{attribute 'c++_compatible'}
// class for implementing IotWebSocetClient functions without exposing them may only be used for ARCommunication_t
FUNCTION_BLOCK ARCommunicationWSExtentionWS_t EXTENDS FB_IotWebSocketClient
VAR_INPUT
END_VAR
VAR_OUTPUT
	lastMessage : STRING(255) := ''; // last recived message
END_VAR
VAR	
	_newMessageAvalable : BOOL := FALSE; // is set true whenever a new message arrives
END_VAR

PROPERTY newMessageAvalable : bool
GET
newMessageAvalable :=  _newMessageAvalable;
END_GET
SET
_newMessageAvalable := newMessageAvalable;
END_SET
END_PROPERTY

{attribute 'TcTypeSystem'}
{attribute 'c++_compatible'}
{attribute 'minimal_input_size' := '4'}
{attribute 'pack_mode' := '4'}
{attribute 'TcRpcEnable'}
METHOD OnWebSocketClose : Global.HRESULT
VAR_INPUT
	statusCode	: UINT;
	content	: Global.PVOID;
	contentLength	: UDINT;
END_VAR
END_METHOD

{attribute 'TcTypeSystem'}
{attribute 'c++_compatible'}
{attribute 'minimal_input_size' := '4'}
{attribute 'pack_mode' := '4'}
{attribute 'TcRpcEnable'}
METHOD OnWebSocketMessage : Global.HRESULT
VAR_INPUT
	content	: Global.PVOID;
	contentLength	: UDINT;
	contentType	: Global.ETcIotWebSocketContentType;
END_VAR
VAR
	ptr : POINTER TO STRING;
END_VAR
// if it isn't text, drop packet
IF  contentType = Global.ETcIotWebSocketContentType.WS_CONTENT_TEXT THEN
		ptr := content;
		THIS^.lastMessage := ptr^;
		THIS^._newMessageAvalable := TRUE;	
END_IF
END_METHOD

{attribute 'TcTypeSystem'}
{attribute 'c++_compatible'}
{attribute 'minimal_input_size' := '4'}
{attribute 'pack_mode' := '4'}
{attribute 'TcRpcEnable'}
METHOD OnWebSocketOpen : Global.HRESULT
VAR_IN_OUT CONSTANT
	webSocketProtocol	: STRING;
	origin	: STRING;
END_VAR
VAR_INPUT
	bPerMessageDeflate	: BOOL;
END_VAR
END_METHOD

{attribute 'TcTypeSystem'}
{attribute 'c++_compatible'}
{attribute 'minimal_input_size' := '4'}
{attribute 'pack_mode' := '4'}
METHOD TcAddRef : UDINT
END_METHOD

{attribute 'TcTypeSystem'}
{attribute 'c++_compatible'}
{attribute 'minimal_input_size' := '4'}
{attribute 'pack_mode' := '4'}
METHOD TcQueryInterface : Global.HRESULT
VAR_INPUT
	iid	: REFERENCE TO Global.IID;
	pipItf	: POINTER TO Global.PVOID;
END_VAR
END_METHOD

{attribute 'TcTypeSystem'}
{attribute 'c++_compatible'}
{attribute 'minimal_input_size' := '4'}
{attribute 'pack_mode' := '4'}
METHOD TcRelease : UDINT
END_METHOD

END_FUNCTION_BLOCK

(* stored: Version 1.1.0.1
   POU ARCommunicationWSExtentionWS_t: Id {b160b582-710e-48ca-a2e1-674bfaf42c51}, SpecialFunc None
   Property newMessageAvalable: Id {60cc030d-e252-40bf-962d-546e21880d27}
   Get Get: Id {89613a16-3d29-4b2d-8a2e-e805c75c660f}
   Set Set: Id {d84cd38f-e2d7-45a5-a66d-f3b744e69d9f}
   Method OnWebSocketClose: Id {83b963f1-cb68-4c4f-839b-6fe0c3279a4b}
   Method OnWebSocketMessage: Id {aafc85e2-e4b6-4b40-a50f-be62207a97c2}
   Method OnWebSocketOpen: Id {84b70aa8-e731-4dfb-b3ce-e492968de315}
   Method TcAddRef: Id {19906943-71ba-4126-b01d-557cf40c9802}
   Method TcQueryInterface: Id {591f8a9a-c7f8-4ed7-bd50-06fbe5fedc76}
   Method TcRelease: Id {02dc99e1-26a5-4db4-a14e-8ac27bc5978f} *)
